// TIA Portal V21 export
// export: Created 2026-07-07T09:15:55.8352405Z, ExportSetting WithReadOnly, DisplayName Totally Integrated Automation Portal, DisplayVersion V21, DisplayName SINAMICS Startdrive Advanced, DisplayVersion V21, DisplayName SINAMICS Startdrive G110M, G120, G120C, G120D, G120P, G115D, DisplayVersion V21, DisplayName SINAMICS Startdrive G130, G150, S120, S150, G200, G220, S200, S210, S220, Innomotics MVD, DisplayVersion V21, DisplayName STEP 7 Professional, DisplayVersion V21, DisplayName STEP 7 Safety, DisplayVersion V21, DisplayName Tech WebApplication, DisplayVersion V21, DisplayName WinCC Basic/Comfort/Advanced, DisplayVersion V21, DisplayName WinCC Professional, DisplayVersion V21, DisplayName WinCC Unified, DisplayVersion V21
Screen "Screen_02_ManualControl"  Nonex480, Template=模板_1
  ScreenLayer 
    TextField "Title" at 20,12 size 760x34  Text="画面 2：手动与调试画面"
    TextField "NavBar" at 20,430 size 760x34  Text="主监控 | 手动调试 | 参数设置 | 报警诊断"
    TextField "Hdr_Item_288" at 20,60 size 360x26  Text="模式控制"
    TextField "Body_Item_304" at 20,84 size 360x96  Text="Manual_Mode | DB1.DBX278.0 | Bool | RW | Auto_Mode | DB1.DBX278.1 | Bool | RW | Emergency_Stop | DB1.DBX278.2 | Bool | RW | Manual_Active | DB1.DBX278.3 | Bool | RO | Auto_Active | DB1.DBX278.4 | Bool | RO"
    TextField "Hdr_Item_320" at 20,190 size 360x26  Text="手动设定输入"
    TextField "Body_Item_336" at 20,214 size 360x166  Text="Manual_q_f_Set | DB1.DBD280 | Real | RW | Manual_q_a_Set | DB1.DBD284 | Real | RW | Manual_q_n_Set | DB1.DBD288 | Real | RW | Manual_q_p_Set | DB1.DBD292 | Real | RW | Manual_q_k_Set | DB1.DBD296 | Real | RW"
    TextField "Hdr_Item_352" at 410,60 size 370x26  Text="联锁与放行"
    TextField "Body_Item_368" at 410,84 size 370x96  Text="Comm_Normal | DB1.DBX300.0 | Bool | RO | Manual_PumpValve_Enable | DB1.DBX300.1 | Bool | RO | Manual_q_f_Selected | DB1.DBD304 | Real | RO | Manual_q_a_Selected | DB1.DBD308 | Real | RO"
    TextField "Hdr_Item_384" at 410,190 size 370x26  Text="执行链路反馈"
    TextField "Body_Item_400" at 410,214 size 370x166  Text="q_f_cmd | DB1.DBD24 | Real | RO | q_a_cmd | DB1.DBD28 | Real | RO | Valve_F_Actual | DB1.DBD32 | Real | RO | Valve_A_Actual | DB1.DBD36 | Real | RO"
